{attribute 'linkalways'} 
{attribute 'no_explicit_call' := 'This FB is a CLASS and must be accessed using methods or properties'}
{attribute 'enable_dynamic_creation'}
FUNCTION_BLOCK Node_F_VN_SubtractContainers EXTENDS VisionNode
VAR
    ipSrcContainer1 : _ITcVnContainer;
    ipSrcContainer2 : _ITcVnContainer;
    ipDestContainer : _ITcVnContainer;
    hrPrev : _HRESULT(S_OK);
    hresult : _HRESULT(S_OK);
END_VAR

METHOD PUBLIC  Clone : I_Node
VAR
    pNode : POINTER TO Node_F_VN_SubtractContainers;
END_VAR
pNode := __NEW(Node_F_VN_SubtractContainers);
Clone := pNode^;
END_METHOD

METHOD FB_init : BOOL
VAR_INPUT
    bInitRetains : BOOL; // if TRUE, the retain variables are initialized (warm start / cold start)
    bInCopyCode : BOOL;  // if TRUE, the instance afterwards gets moved into the copy code (online change)
END_VAR
AddInput('ipSrcContainer1', ipSrcContainer1);
AddInput('ipSrcContainer2', ipSrcContainer2);
AddInput('hrPrev', hrPrev);
AddOutput('ipDestContainer', ipDestContainer);
AddOutput('hresult',hresult);
END_METHOD

METHOD PROTECTED OnExecute
hresult.Value := F_VN_SubtractContainers(
    ipSrcContainer1 := ipSrcContainer1.Value,
    ipSrcContainer2 := ipSrcContainer2.Value,
    ipDestContainer := ipDestContainer.Value,
    hrPrev:= hrPrev.Value);
END_METHOD

METHOD PUBLIC PreExecutionCheck
VAR_INPUT
    Check : I_PreExecutionChecks;
END_VAR
Check.IsTrue(ipSrcContainer1.IsValid, 'ipSrcContainer1 must be a valid container');
Check.IsTrue(ipSrcContainer2.IsValid, 'ipSrcContainer2 must be a valid container');
Check.IsTrue(ContainersHaveMatchingTypes(ipSrcContainer1.Value, ipSrcContainer2.Value), 'Source containers must have matching types');
Check.IsTrue(ContainersHaveMatchingNumberOfElements(ipSrcContainer1.Value, ipSrcContainer2.Value), 'Source containers must contain the same number of elements');
END_METHOD

END_FUNCTION_BLOCK

(* stored: Version 1.1.0.1, ProductVersion 3.1.4024.15
   POU Node_F_VN_SubtractContainers: Id {942960a2-4ab5-09ca-3807-b84ce427e99e}, SpecialFunc None
   Folder Constructor: Id {8cca6cda-b32a-03f6-07c9-5fbb878a184d}
   Method Clone: Id {6c0889c1-4668-063e-3140-03ee5fb76e0c}
   Method FB_init: Id {2fc80d78-9a79-04ae-33c9-b6bed3ae57d5}
   Method OnExecute: Id {9f12cddd-0282-0aa5-2abb-beb43ecad23b}
   Method PreExecutionCheck: Id {9f3885b7-5e4b-0b30-0a31-fbf4cbab80d6} *)
